(* Logix 5000 project; controller NSH_PLC2 vendor 1 type 14 code 167 rev 32.14; software revision 32.03; part 5 of 6 *)
(* tags used below, declared in another part *)
   AFI : BOOL;   // Always False
   AOI_MCC4_3E_ToPLC1 : E300ToMotor;
   AOI_MCC4_3G_ToPLC1 : E300ToMotor;
   AOI_MCC4_3J_ToPLC1 : E300ToMotor;
   AOI_MCC4_3L_ToPLC1 : E300ToMotor;
   AOI_MCC4_4A_ToPLC1 : E300ToMotor;
   AOI_MCC4_4C_ToPLC1 : E300ToMotor;
   AOI_MCC4_4E_ToPLC1 : E300ToMotor;
   AOI_MCC4_4G_ToPLC1 : E300ToMotor;
   AOI_MCC4_4J_ToPLC1 : E300ToMotor;
   AOI_MCC4_4L_ToPLC1 : E300ToMotor;
   AOI_MCC4_5A_ToPLC1 : E300ToMotor;
   AOI_MCC4_5C_ToPLC1 : E300ToMotor;
   AOI_PLC1_To_MCC2_10A : MotorToE300;
   AOI_PLC1_To_MCC2_10C : MotorToE300;
   AOI_PLC1_To_MCC2_10E : MotorToE300;
   AOI_PLC1_To_MCC2_10G : MotorToE300;
   AOI_PLC1_To_MCC2_10J : MotorToE300;
   AOI_PLC1_To_MCC2_10L : MotorToE300;
   AOI_PLC1_To_MCC2_11A : MotorToE300;
   AOI_PLC1_To_MCC2_11C : MotorToE300;
   AOI_PLC1_To_MCC2_11E : MotorToE300;
   AOI_PLC1_To_MCC2_11G : MotorToE300;
   AOI_PLC1_To_MCC2_11J : MotorToE300;
   AOI_PLC1_To_MCC2_11L : MotorToE300;
   AOI_PLC1_To_MCC2_12A : MotorToE300;
   AOI_PLC1_To_MCC2_12C : MotorToE300;
   AOI_PLC1_To_MCC2_12E : MotorToE300;
   AOI_PLC1_To_MCC2_12G : MotorToE300;
   AOI_PLC1_To_MCC2_12J : MotorToE300;
   AOI_PLC1_To_MCC2_12L : MotorToE300;
   AOI_PLC1_To_MCC2_13A : MotorToE300;
   AOI_PLC1_To_MCC2_13C : MotorToE300;
   AOI_PLC1_To_MCC2_13E : MotorToE300;
   AOI_PLC1_To_MCC2_13G : MotorToE300;
   AOI_PLC1_To_MCC2_13J : MotorToE300;
   AOI_PLC1_To_MCC2_14A : MotorToE300;
   AOI_PLC1_To_MCC2_14C : MotorToE300;
   AOI_PLC1_To_MCC2_14E : MotorToE300;
   AOI_PLC1_To_MCC2_14G : MotorToE300;
   AOI_PLC1_To_MCC2_14J : MotorToE300;
   AOI_PLC1_To_MCC2_14L : MotorToE300;
   AOI_PLC1_To_MCC2_15A : MotorToE300;
   AOI_PLC1_To_MCC2_15C : MotorToE300;
   AOI_PLC1_To_MCC2_15E : MotorToE300;
   AOI_PLC1_To_MCC2_15G : MotorToE300;
   AOI_PLC1_To_MCC2_15J : MotorToE300;
   AOI_PLC1_To_MCC2_15L : MotorToE300;
   AOI_PLC1_To_MCC2_16A : MotorToE300;
   AOI_PLC1_To_MCC2_16C : MotorToE300;
   AOI_PLC1_To_MCC2_16E : MotorToE300;
   AOI_PLC1_To_MCC2_16G : MotorToE300;
   AOI_PLC1_To_MCC2_16J : MotorToE300;
   AOI_PLC1_To_MCC2_16L : MotorToE300;
   AOI_PLC1_To_MCC2_17A : MotorToE300;
   AOI_PLC1_To_MCC2_17C : MotorToE300;
   AOI_PLC1_To_MCC2_17E : MotorToE300;
   AOI_PLC1_To_MCC2_17G : MotorToE300;
   AOI_PLC1_To_MCC2_17J : MotorToE300;
   AOI_PLC1_To_MCC2_18A : MotorToE300;
   AOI_PLC1_To_MCC2_18C : MotorToE300;
   AOI_PLC1_To_MCC2_18E : MotorToE300;
   AOI_PLC1_To_MCC2_18G : MotorToE300;
   AOI_PLC1_To_MCC2_18J : MotorToE300;
   AOI_PLC1_To_MCC2_18L : MotorToE300;
   AOI_PLC1_To_MCC2_19A : MotorToE300;
   AOI_PLC1_To_MCC2_19C : MotorToE300;
   AOI_PLC1_To_MCC2_19E : MotorToE300;
   AOI_PLC1_To_MCC2_19G : MotorToE300;
   AOI_PLC1_To_MCC2_19J : MotorToE300;
   AOI_PLC1_To_MCC2_19L : MotorToE300;
   AOI_PLC1_To_MCC2_20C : MotorToE300;
   AOI_PLC1_To_MCC2_20E : MotorToE300;
   AOI_PLC1_To_MCC2_20G : MotorToE300;
   AOI_PLC1_To_MCC2_20J : MotorToE300;
   AOI_PLC1_To_MCC2_21A : MotorToE300;
   AOI_PLC1_To_MCC2_21C : MotorToE300;
   AOI_PLC1_To_MCC2_21E : MotorToE300;
   AOI_PLC1_To_MCC2_21G : MotorToPF525;
   AOI_PLC1_To_MCC2_21K : MotorToPF525;
   AOI_PLC1_To_MCC2_2A : MotorToPF525;   // Motor From PLC1 to PF525 AOI
   AOI_PLC1_To_MCC2_2D : MotorToPF525;
   AOI_PLC1_To_MCC2_2G : MotorToPF525;
   AOI_PLC1_To_MCC2_2K : MotorToPF525;
   AOI_PLC1_To_MCC2_3A : MotorToE300;
   AOI_PLC1_To_MCC2_3C : MotorToE300;
   AOI_PLC1_To_MCC2_3E : MotorToE300;
   AOI_PLC1_To_MCC2_3G : MotorToE300;
   AOI_PLC1_To_MCC2_3J : MotorToE300;
   AOI_PLC1_To_MCC2_3L : MotorToE300;
   AOI_PLC1_To_MCC2_4A : MotorToE300;
   AOI_PLC1_To_MCC2_4C : MotorToE300;
   AOI_PLC1_To_MCC2_4E : MotorToE300;
   AOI_PLC1_To_MCC2_4G : MotorToE300;
   AOI_PLC1_To_MCC2_4J : MotorToE300;
   AOI_PLC1_To_MCC2_4L : MotorToE300;
   AOI_PLC1_To_MCC2_5A : MotorToE300;
   AOI_PLC1_To_MCC2_5C : MotorToE300;
   AOI_PLC1_To_MCC2_5E : MotorToE300;
   AOI_PLC1_To_MCC2_5G : MotorToE300;
   AOI_PLC1_To_MCC2_5J : MotorToE300;
   AOI_PLC1_To_MCC2_6A : MotorToE300;
   AOI_PLC1_To_MCC2_6C : MotorToE300;
   AOI_PLC1_To_MCC2_6E : MotorToE300;
   AOI_PLC1_To_MCC2_6G : MotorToE300;
   AOI_PLC1_To_MCC2_6J : MotorToE300;
   AOI_PLC1_To_MCC2_6L : MotorToE300;
   AOI_PLC1_To_MCC2_7A : MotorToE300;
   AOI_PLC1_To_MCC2_7D : MotorToE300;
   AOI_PLC1_To_MCC2_7G : MotorToE300;
   AOI_PLC1_To_MCC2_7K : MotorToE300;
   AOI_PLC1_To_MCC2_8B : MotorToE300;
   AOI_PLC1_To_MCC2_8D : MotorToE300;
   AOI_PLC1_To_MCC2_8F : MotorToE300;
   AOI_PLC1_To_MCC2_8H : MotorToE300;
   AOI_PLC1_To_MCC2_8K : MotorToE300;
   AOI_PLC1_To_MCC2_9D : MotorToE300;
   AOI_PLC1_To_MCC2_9F : MotorToE300;
   AOI_PLC1_To_MCC2_9H : MotorToPF525;
   AOI_PLC1_To_MCC3_2A : MotorToPF525;
   AOI_PLC1_To_MCC3_2D : MotorToPF525;
   AOI_PLC1_To_MCC3_2G : MotorToPF525;
   AOI_PLC1_To_MCC3_2K : MotorToPF525;
   AOI_PLC1_To_MCC3_3A : MotorToPF525;
   AOI_PLC1_To_MCC3_3D : MotorToPF525;
   AOI_PLC1_To_MCC3_3G : MotorToPF525;
   AOI_PLC1_To_MCC3_3K : MotorToPF525;
   AOI_PLC1_To_MCC3_4A : MotorToPF525;
   AOI_PLC1_To_MCC3_4D : MotorToPF525;
   AOI_PLC1_To_MCC3_4G : MotorToPF525;
   AOI_PLC1_To_MCC3_4K : MotorToPF525;
   AOI_PLC1_To_MCC3_5A : MotorToPF525;
   AOI_PLC1_To_MCC3_5D : MotorToPF525;
   AOI_PLC1_To_MCC3_5G : MotorToPF525;
   AOI_PLC1_To_MCC3_5K : MotorToPF525;
   AOI_PLC1_To_MCC3_6A : MotorToPF525;
   AOI_PLC1_To_MCC3_6D : MotorToPF525;
   AOI_PLC1_To_MCC3_6G : MotorToE300;
   AOI_PLC1_To_MCC3_6J : MotorToE300;
   Const_4000_Hex : INT;   // Constant #16:4000, Entry Status Communicating
   GSV_EntryStatus : INT;   // GSV Entry Status, shold be #16:4000
   MCC4_3E_CommsOK : BOOL;   // Communications with AOP OK
   MCC4_3G_CommsOK : BOOL;   // Communications with AOP OK
   MCC4_3J_CommsOK : BOOL;   // Communications with AOP OK
   MCC4_3L_CommsOK : BOOL;   // Communications with AOP OK
   MCC4_4A_CommsOK : BOOL;   // Communications with AOP OK
   MCC4_4C_CommsOK : BOOL;   // Communications with AOP OK
   MCC4_4E_CommsOK : BOOL;   // Communications with AOP OK
   MCC4_4G_CommsOK : BOOL;   // Communications with AOP OK
   MCC4_4J_CommsOK : BOOL;   // Communications with AOP OK
   MCC4_4L_CommsOK : BOOL;   // Communications with AOP OK
   MCC4_5A_CommsOK : BOOL;   // Communications with AOP OK
   MCC4_5C_CommsOK : BOOL;   // Communications with AOP OK
   MotorsControlTag : MotorsControlUDT;   // Only Instance of UDT
   MotorsStatusTag : MotorsStatusUDT;   // Only Instance of UDT
   MSG_ReadSpacing_T : TIMER;   // Read MCC2 & MCC3 Motor Commands From PLC1 Spacing Timer
   OKToRunMotors : BOOL;   // Messages from PLC1 Ok, OK to run
   ReadMotorError_CTR : COUNTER;   // Read Message form PLC1 Error Counter
   ReadMotorsFromPLC1 : MESSAGE;   // Read from PLC1, MotorsToPLC2
   ReadMotorsFromPLC1_DOS : BOOL;   // Read Motors from PLC1 Done One Shot
(* MainProgram, continued *)

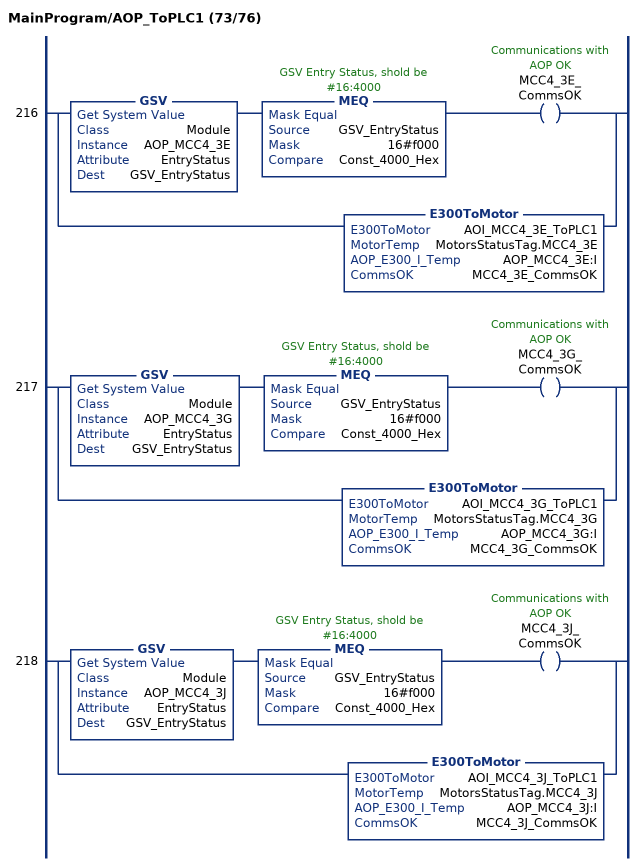
   216: [GSV(Module,AOP_MCC4_3E,EntryStatus,GSV_EntryStatus) MEQ(GSV_EntryStatus,16#f000,Const_4000_Hex) OTE(MCC4_3E_CommsOK) ,E300ToMotor(AOI_MCC4_3E_ToPLC1,MotorsStatusTag.MCC4_3E,AOP_MCC4_3E:I,MCC4_3E_CommsOK) ];
   217: [GSV(Module,AOP_MCC4_3G,EntryStatus,GSV_EntryStatus) MEQ(GSV_EntryStatus,16#f000,Const_4000_Hex) OTE(MCC4_3G_CommsOK) ,E300ToMotor(AOI_MCC4_3G_ToPLC1,MotorsStatusTag.MCC4_3G,AOP_MCC4_3G:I,MCC4_3G_CommsOK) ];
   218: [GSV(Module,AOP_MCC4_3J,EntryStatus,GSV_EntryStatus) MEQ(GSV_EntryStatus,16#f000,Const_4000_Hex) OTE(MCC4_3J_CommsOK) ,E300ToMotor(AOI_MCC4_3J_ToPLC1,MotorsStatusTag.MCC4_3J,AOP_MCC4_3J:I,MCC4_3J_CommsOK) ];
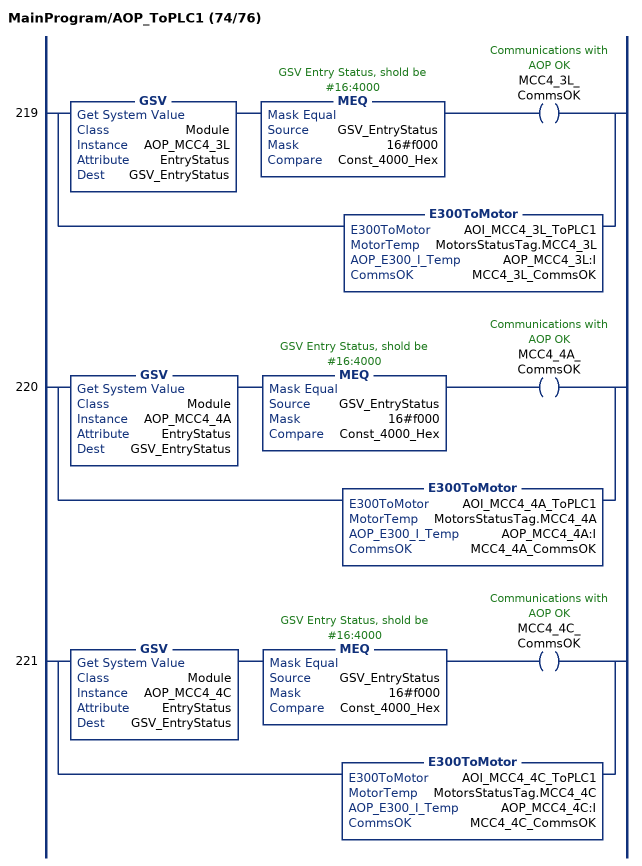
   219: [GSV(Module,AOP_MCC4_3L,EntryStatus,GSV_EntryStatus) MEQ(GSV_EntryStatus,16#f000,Const_4000_Hex) OTE(MCC4_3L_CommsOK) ,E300ToMotor(AOI_MCC4_3L_ToPLC1,MotorsStatusTag.MCC4_3L,AOP_MCC4_3L:I,MCC4_3L_CommsOK) ];
   220: [GSV(Module,AOP_MCC4_4A,EntryStatus,GSV_EntryStatus) MEQ(GSV_EntryStatus,16#f000,Const_4000_Hex) OTE(MCC4_4A_CommsOK) ,E300ToMotor(AOI_MCC4_4A_ToPLC1,MotorsStatusTag.MCC4_4A,AOP_MCC4_4A:I,MCC4_4A_CommsOK) ];
   221: [GSV(Module,AOP_MCC4_4C,EntryStatus,GSV_EntryStatus) MEQ(GSV_EntryStatus,16#f000,Const_4000_Hex) OTE(MCC4_4C_CommsOK) ,E300ToMotor(AOI_MCC4_4C_ToPLC1,MotorsStatusTag.MCC4_4C,AOP_MCC4_4C:I,MCC4_4C_CommsOK) ];
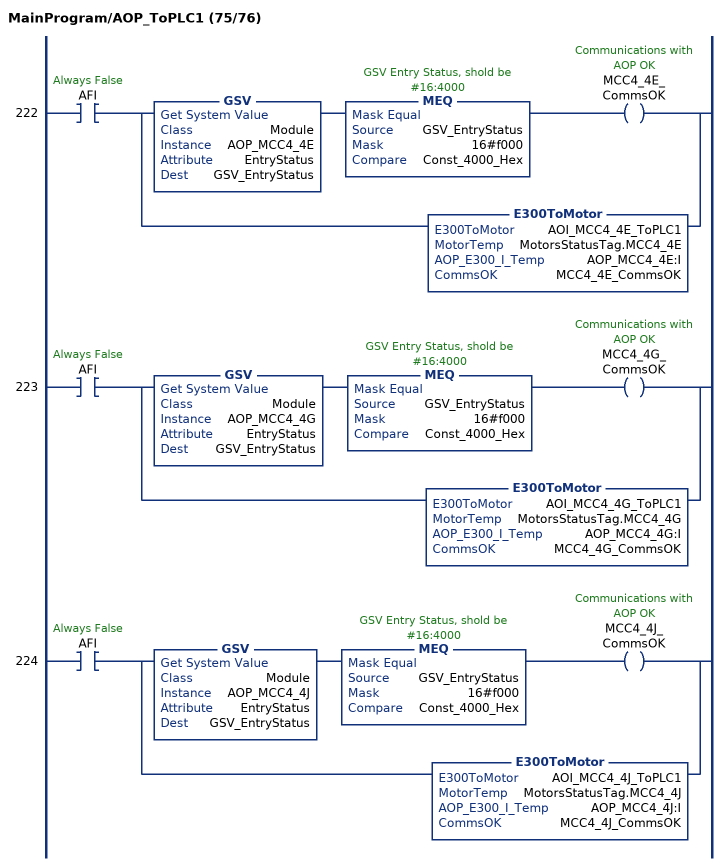
   222: XIC(AFI)[GSV(Module,AOP_MCC4_4E,EntryStatus,GSV_EntryStatus) MEQ(GSV_EntryStatus,16#f000,Const_4000_Hex) OTE(MCC4_4E_CommsOK) ,E300ToMotor(AOI_MCC4_4E_ToPLC1,MotorsStatusTag.MCC4_4E,AOP_MCC4_4E:I,MCC4_4E_CommsOK) ];
   223: XIC(AFI)[GSV(Module,AOP_MCC4_4G,EntryStatus,GSV_EntryStatus) MEQ(GSV_EntryStatus,16#f000,Const_4000_Hex) OTE(MCC4_4G_CommsOK) ,E300ToMotor(AOI_MCC4_4G_ToPLC1,MotorsStatusTag.MCC4_4G,AOP_MCC4_4G:I,MCC4_4G_CommsOK) ];
   224: XIC(AFI)[GSV(Module,AOP_MCC4_4J,EntryStatus,GSV_EntryStatus) MEQ(GSV_EntryStatus,16#f000,Const_4000_Hex) OTE(MCC4_4J_CommsOK) ,E300ToMotor(AOI_MCC4_4J_ToPLC1,MotorsStatusTag.MCC4_4J,AOP_MCC4_4J:I,MCC4_4J_CommsOK) ];
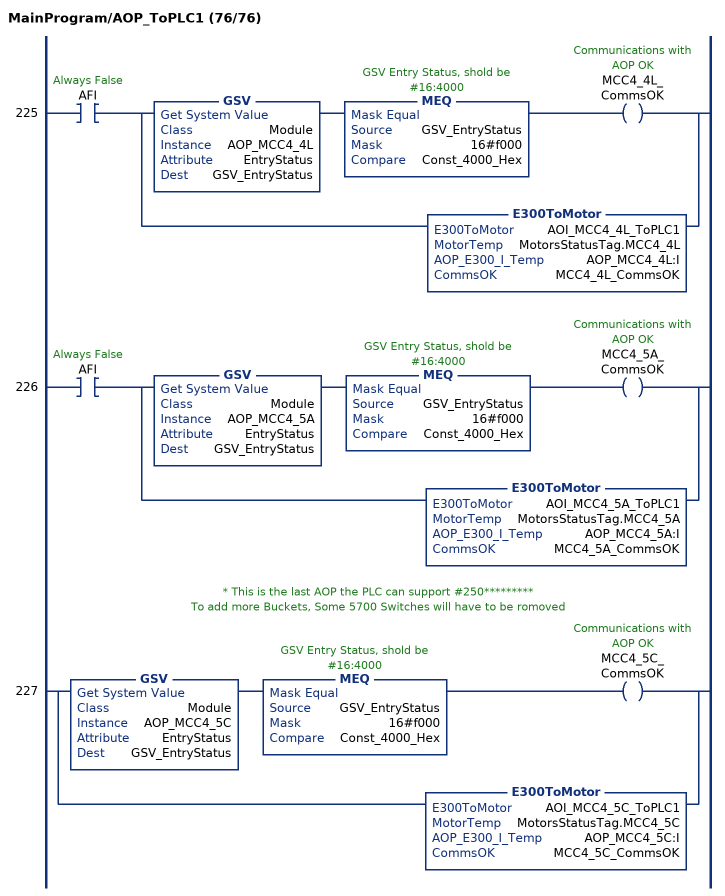
   225: XIC(AFI)[GSV(Module,AOP_MCC4_4L,EntryStatus,GSV_EntryStatus) MEQ(GSV_EntryStatus,16#f000,Const_4000_Hex) OTE(MCC4_4L_CommsOK) ,E300ToMotor(AOI_MCC4_4L_ToPLC1,MotorsStatusTag.MCC4_4L,AOP_MCC4_4L:I,MCC4_4L_CommsOK) ];
   226: XIC(AFI)[GSV(Module,AOP_MCC4_5A,EntryStatus,GSV_EntryStatus) MEQ(GSV_EntryStatus,16#f000,Const_4000_Hex) OTE(MCC4_5A_CommsOK) ,E300ToMotor(AOI_MCC4_5A_ToPLC1,MotorsStatusTag.MCC4_5A,AOP_MCC4_5A:I,MCC4_5A_CommsOK) ];
   // * This is the last AOP the PLC can support #250*********
   // To add more Buckets, Some 5700 Switches will have to be romoved
   227: [GSV(Module,AOP_MCC4_5C,EntryStatus,GSV_EntryStatus) MEQ(GSV_EntryStatus,16#f000,Const_4000_Hex) OTE(MCC4_5C_CommsOK) ,E300ToMotor(AOI_MCC4_5C_ToPLC1,MotorsStatusTag.MCC4_5C,AOP_MCC4_5C:I,MCC4_5C_CommsOK) ];
END_ROUTINE

ROUTINE MainRoutine   (* ladder *)
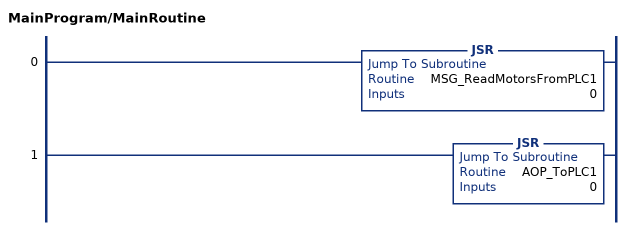
   0: JSR(MSG_ReadMotorsFromPLC1,0);
   1: JSR(AOP_ToPLC1,0);
END_ROUTINE

ROUTINE MSG_ReadMotorsFromPLC1   (* ladder *)
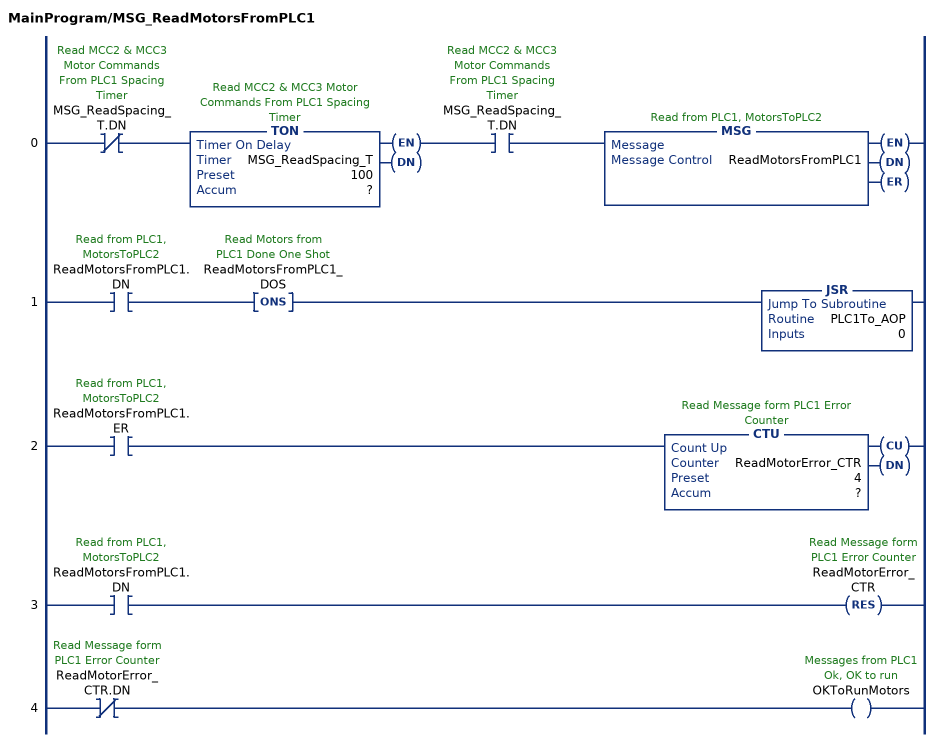
   0: XIO(MSG_ReadSpacing_T.DN)TON(MSG_ReadSpacing_T,?,?)XIC(MSG_ReadSpacing_T.DN)MSG(ReadMotorsFromPLC1);
   1: XIC(ReadMotorsFromPLC1.DN)ONS(ReadMotorsFromPLC1_DOS)JSR(PLC1To_AOP,0);
   2: XIC(ReadMotorsFromPLC1.ER)CTU(ReadMotorError_CTR,?,?);
   3: XIC(ReadMotorsFromPLC1.DN)RES(ReadMotorError_CTR);
   4: XIO(ReadMotorError_CTR.DN)OTE(OKToRunMotors);
END_ROUTINE

ROUTINE PLC1To_AOP   (* ladder *)
// Send Command Data from PLC#1 to AOPs
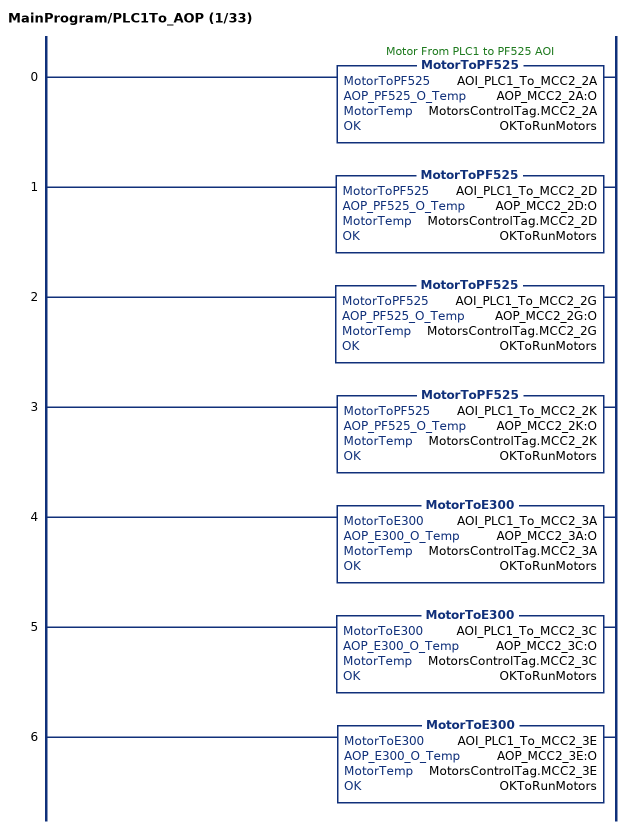
   0: MotorToPF525(AOI_PLC1_To_MCC2_2A,AOP_MCC2_2A:O,MotorsControlTag.MCC2_2A,OKToRunMotors);
   1: MotorToPF525(AOI_PLC1_To_MCC2_2D,AOP_MCC2_2D:O,MotorsControlTag.MCC2_2D,OKToRunMotors);
   2: MotorToPF525(AOI_PLC1_To_MCC2_2G,AOP_MCC2_2G:O,MotorsControlTag.MCC2_2G,OKToRunMotors);
   3: MotorToPF525(AOI_PLC1_To_MCC2_2K,AOP_MCC2_2K:O,MotorsControlTag.MCC2_2K,OKToRunMotors);
   4: MotorToE300(AOI_PLC1_To_MCC2_3A,AOP_MCC2_3A:O,MotorsControlTag.MCC2_3A,OKToRunMotors);
   5: MotorToE300(AOI_PLC1_To_MCC2_3C,AOP_MCC2_3C:O,MotorsControlTag.MCC2_3C,OKToRunMotors);
   6: MotorToE300(AOI_PLC1_To_MCC2_3E,AOP_MCC2_3E:O,MotorsControlTag.MCC2_3E,OKToRunMotors);
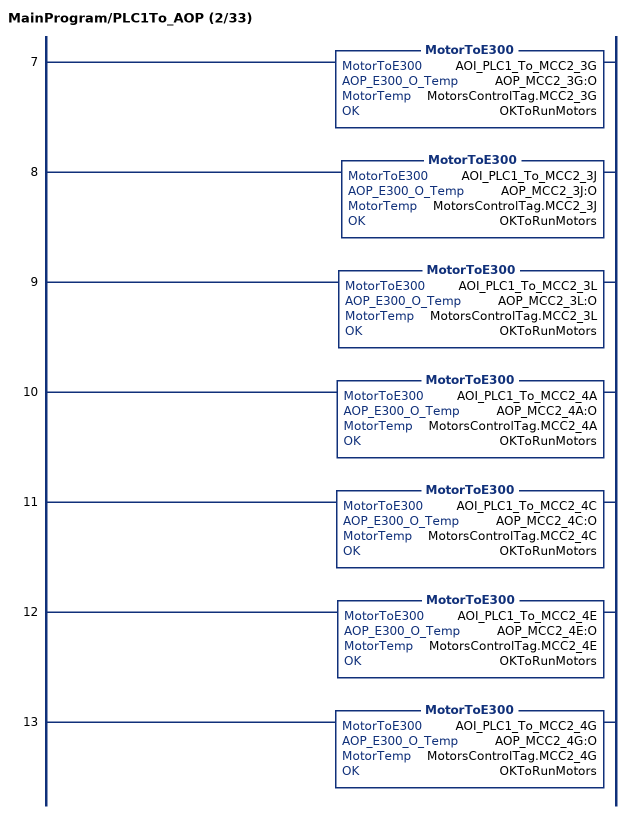
   7: MotorToE300(AOI_PLC1_To_MCC2_3G,AOP_MCC2_3G:O,MotorsControlTag.MCC2_3G,OKToRunMotors);
   8: MotorToE300(AOI_PLC1_To_MCC2_3J,AOP_MCC2_3J:O,MotorsControlTag.MCC2_3J,OKToRunMotors);
   9: MotorToE300(AOI_PLC1_To_MCC2_3L,AOP_MCC2_3L:O,MotorsControlTag.MCC2_3L,OKToRunMotors);
   10: MotorToE300(AOI_PLC1_To_MCC2_4A,AOP_MCC2_4A:O,MotorsControlTag.MCC2_4A,OKToRunMotors);
   11: MotorToE300(AOI_PLC1_To_MCC2_4C,AOP_MCC2_4C:O,MotorsControlTag.MCC2_4C,OKToRunMotors);
   12: MotorToE300(AOI_PLC1_To_MCC2_4E,AOP_MCC2_4E:O,MotorsControlTag.MCC2_4E,OKToRunMotors);
   13: MotorToE300(AOI_PLC1_To_MCC2_4G,AOP_MCC2_4G:O,MotorsControlTag.MCC2_4G,OKToRunMotors);
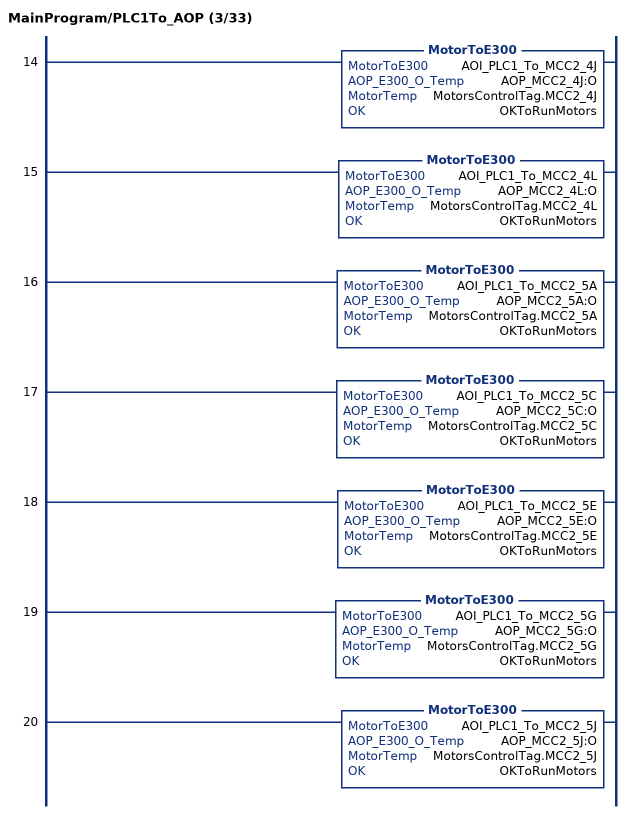
   14: MotorToE300(AOI_PLC1_To_MCC2_4J,AOP_MCC2_4J:O,MotorsControlTag.MCC2_4J,OKToRunMotors);
   15: MotorToE300(AOI_PLC1_To_MCC2_4L,AOP_MCC2_4L:O,MotorsControlTag.MCC2_4L,OKToRunMotors);
   16: MotorToE300(AOI_PLC1_To_MCC2_5A,AOP_MCC2_5A:O,MotorsControlTag.MCC2_5A,OKToRunMotors);
   17: MotorToE300(AOI_PLC1_To_MCC2_5C,AOP_MCC2_5C:O,MotorsControlTag.MCC2_5C,OKToRunMotors);
   18: MotorToE300(AOI_PLC1_To_MCC2_5E,AOP_MCC2_5E:O,MotorsControlTag.MCC2_5E,OKToRunMotors);
   19: MotorToE300(AOI_PLC1_To_MCC2_5G,AOP_MCC2_5G:O,MotorsControlTag.MCC2_5G,OKToRunMotors);
   20: MotorToE300(AOI_PLC1_To_MCC2_5J,AOP_MCC2_5J:O,MotorsControlTag.MCC2_5J,OKToRunMotors);
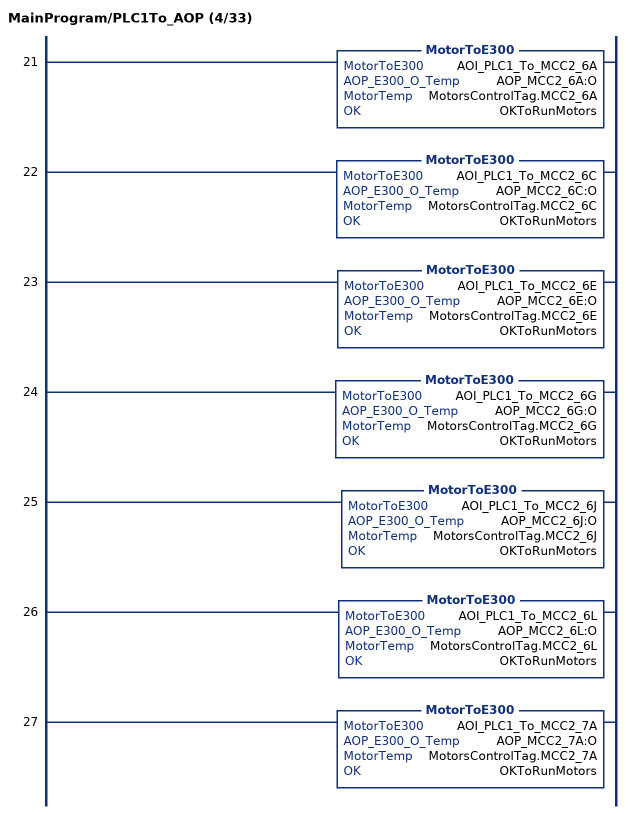
   21: MotorToE300(AOI_PLC1_To_MCC2_6A,AOP_MCC2_6A:O,MotorsControlTag.MCC2_6A,OKToRunMotors);
   22: MotorToE300(AOI_PLC1_To_MCC2_6C,AOP_MCC2_6C:O,MotorsControlTag.MCC2_6C,OKToRunMotors);
   23: MotorToE300(AOI_PLC1_To_MCC2_6E,AOP_MCC2_6E:O,MotorsControlTag.MCC2_6E,OKToRunMotors);
   24: MotorToE300(AOI_PLC1_To_MCC2_6G,AOP_MCC2_6G:O,MotorsControlTag.MCC2_6G,OKToRunMotors);
   25: MotorToE300(AOI_PLC1_To_MCC2_6J,AOP_MCC2_6J:O,MotorsControlTag.MCC2_6J,OKToRunMotors);
   26: MotorToE300(AOI_PLC1_To_MCC2_6L,AOP_MCC2_6L:O,MotorsControlTag.MCC2_6L,OKToRunMotors);
   27: MotorToE300(AOI_PLC1_To_MCC2_7A,AOP_MCC2_7A:O,MotorsControlTag.MCC2_7A,OKToRunMotors);
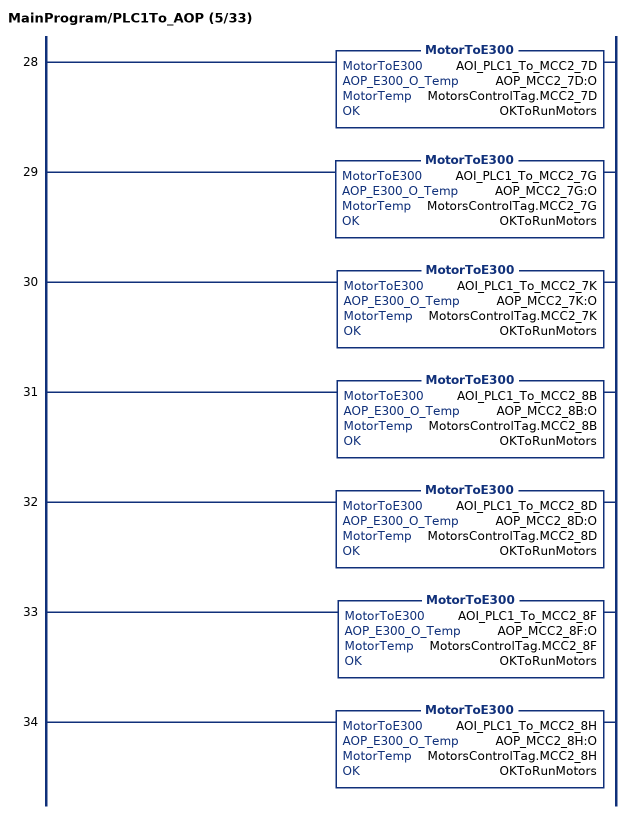
   28: MotorToE300(AOI_PLC1_To_MCC2_7D,AOP_MCC2_7D:O,MotorsControlTag.MCC2_7D,OKToRunMotors);
   29: MotorToE300(AOI_PLC1_To_MCC2_7G,AOP_MCC2_7G:O,MotorsControlTag.MCC2_7G,OKToRunMotors);
   30: MotorToE300(AOI_PLC1_To_MCC2_7K,AOP_MCC2_7K:O,MotorsControlTag.MCC2_7K,OKToRunMotors);
   31: MotorToE300(AOI_PLC1_To_MCC2_8B,AOP_MCC2_8B:O,MotorsControlTag.MCC2_8B,OKToRunMotors);
   32: MotorToE300(AOI_PLC1_To_MCC2_8D,AOP_MCC2_8D:O,MotorsControlTag.MCC2_8D,OKToRunMotors);
   33: MotorToE300(AOI_PLC1_To_MCC2_8F,AOP_MCC2_8F:O,MotorsControlTag.MCC2_8F,OKToRunMotors);
   34: MotorToE300(AOI_PLC1_To_MCC2_8H,AOP_MCC2_8H:O,MotorsControlTag.MCC2_8H,OKToRunMotors);
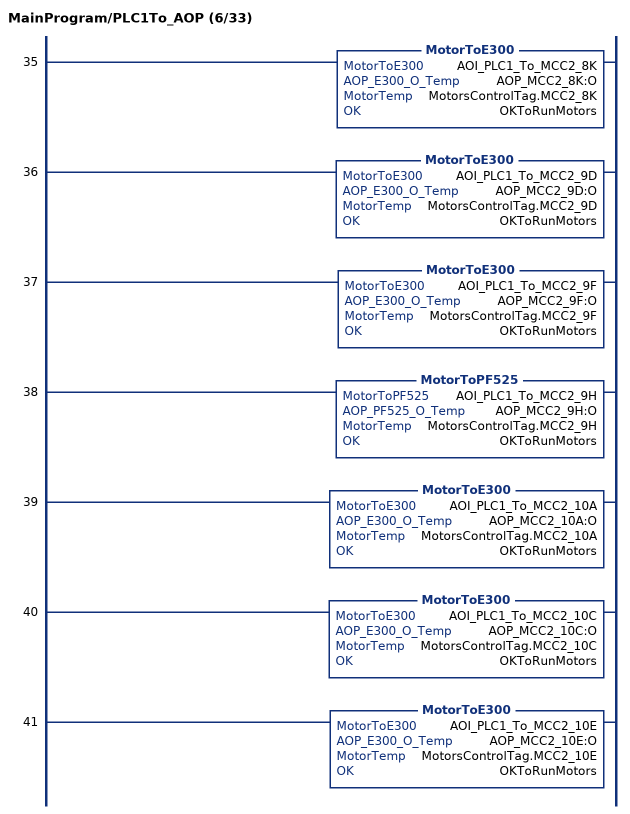
   35: MotorToE300(AOI_PLC1_To_MCC2_8K,AOP_MCC2_8K:O,MotorsControlTag.MCC2_8K,OKToRunMotors);
   36: MotorToE300(AOI_PLC1_To_MCC2_9D,AOP_MCC2_9D:O,MotorsControlTag.MCC2_9D,OKToRunMotors);
   37: MotorToE300(AOI_PLC1_To_MCC2_9F,AOP_MCC2_9F:O,MotorsControlTag.MCC2_9F,OKToRunMotors);
   38: MotorToPF525(AOI_PLC1_To_MCC2_9H,AOP_MCC2_9H:O,MotorsControlTag.MCC2_9H,OKToRunMotors);
   39: MotorToE300(AOI_PLC1_To_MCC2_10A,AOP_MCC2_10A:O,MotorsControlTag.MCC2_10A,OKToRunMotors);
   40: MotorToE300(AOI_PLC1_To_MCC2_10C,AOP_MCC2_10C:O,MotorsControlTag.MCC2_10C,OKToRunMotors);
   41: MotorToE300(AOI_PLC1_To_MCC2_10E,AOP_MCC2_10E:O,MotorsControlTag.MCC2_10E,OKToRunMotors);
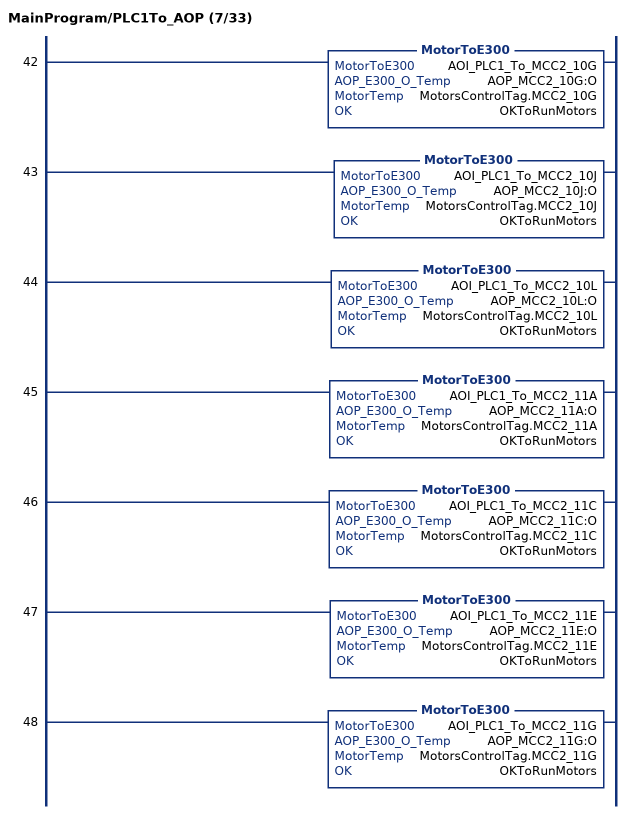
   42: MotorToE300(AOI_PLC1_To_MCC2_10G,AOP_MCC2_10G:O,MotorsControlTag.MCC2_10G,OKToRunMotors);
   43: MotorToE300(AOI_PLC1_To_MCC2_10J,AOP_MCC2_10J:O,MotorsControlTag.MCC2_10J,OKToRunMotors);
   44: MotorToE300(AOI_PLC1_To_MCC2_10L,AOP_MCC2_10L:O,MotorsControlTag.MCC2_10L,OKToRunMotors);
   45: MotorToE300(AOI_PLC1_To_MCC2_11A,AOP_MCC2_11A:O,MotorsControlTag.MCC2_11A,OKToRunMotors);
   46: MotorToE300(AOI_PLC1_To_MCC2_11C,AOP_MCC2_11C:O,MotorsControlTag.MCC2_11C,OKToRunMotors);
   47: MotorToE300(AOI_PLC1_To_MCC2_11E,AOP_MCC2_11E:O,MotorsControlTag.MCC2_11E,OKToRunMotors);
   48: MotorToE300(AOI_PLC1_To_MCC2_11G,AOP_MCC2_11G:O,MotorsControlTag.MCC2_11G,OKToRunMotors);
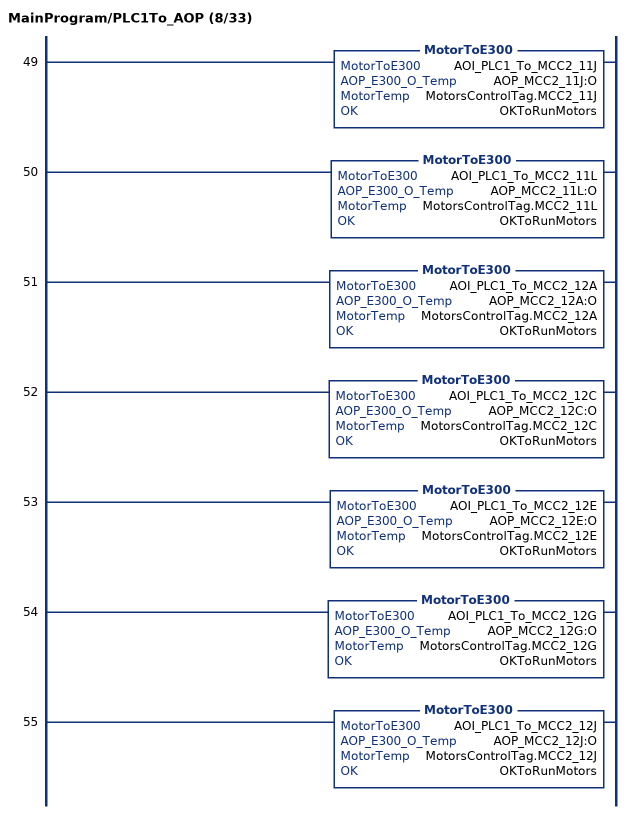
   49: MotorToE300(AOI_PLC1_To_MCC2_11J,AOP_MCC2_11J:O,MotorsControlTag.MCC2_11J,OKToRunMotors);
   50: MotorToE300(AOI_PLC1_To_MCC2_11L,AOP_MCC2_11L:O,MotorsControlTag.MCC2_11L,OKToRunMotors);
   51: MotorToE300(AOI_PLC1_To_MCC2_12A,AOP_MCC2_12A:O,MotorsControlTag.MCC2_12A,OKToRunMotors);
   52: MotorToE300(AOI_PLC1_To_MCC2_12C,AOP_MCC2_12C:O,MotorsControlTag.MCC2_12C,OKToRunMotors);
   53: MotorToE300(AOI_PLC1_To_MCC2_12E,AOP_MCC2_12E:O,MotorsControlTag.MCC2_12E,OKToRunMotors);
   54: MotorToE300(AOI_PLC1_To_MCC2_12G,AOP_MCC2_12G:O,MotorsControlTag.MCC2_12G,OKToRunMotors);
   55: MotorToE300(AOI_PLC1_To_MCC2_12J,AOP_MCC2_12J:O,MotorsControlTag.MCC2_12J,OKToRunMotors);
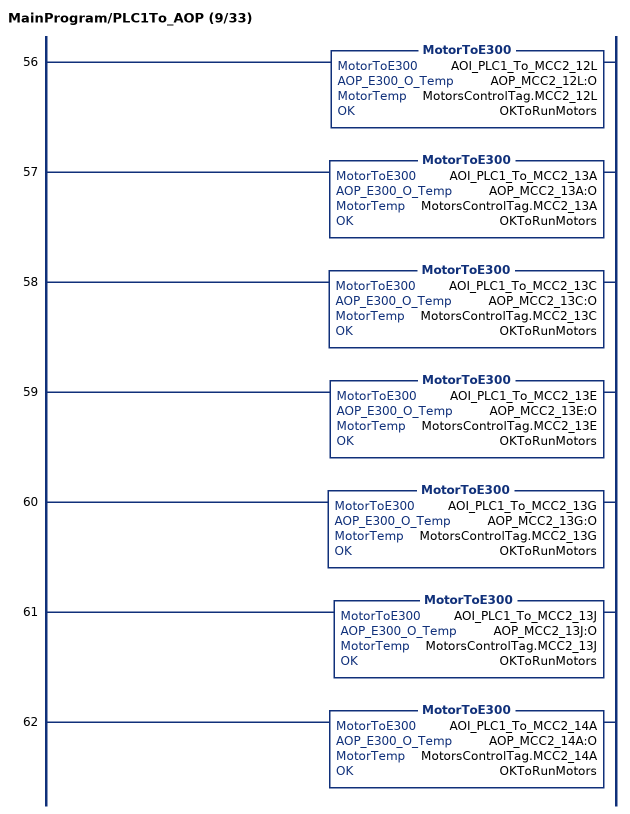
   56: MotorToE300(AOI_PLC1_To_MCC2_12L,AOP_MCC2_12L:O,MotorsControlTag.MCC2_12L,OKToRunMotors);
   57: MotorToE300(AOI_PLC1_To_MCC2_13A,AOP_MCC2_13A:O,MotorsControlTag.MCC2_13A,OKToRunMotors);
   58: MotorToE300(AOI_PLC1_To_MCC2_13C,AOP_MCC2_13C:O,MotorsControlTag.MCC2_13C,OKToRunMotors);
   59: MotorToE300(AOI_PLC1_To_MCC2_13E,AOP_MCC2_13E:O,MotorsControlTag.MCC2_13E,OKToRunMotors);
   60: MotorToE300(AOI_PLC1_To_MCC2_13G,AOP_MCC2_13G:O,MotorsControlTag.MCC2_13G,OKToRunMotors);
   61: MotorToE300(AOI_PLC1_To_MCC2_13J,AOP_MCC2_13J:O,MotorsControlTag.MCC2_13J,OKToRunMotors);
   62: MotorToE300(AOI_PLC1_To_MCC2_14A,AOP_MCC2_14A:O,MotorsControlTag.MCC2_14A,OKToRunMotors);
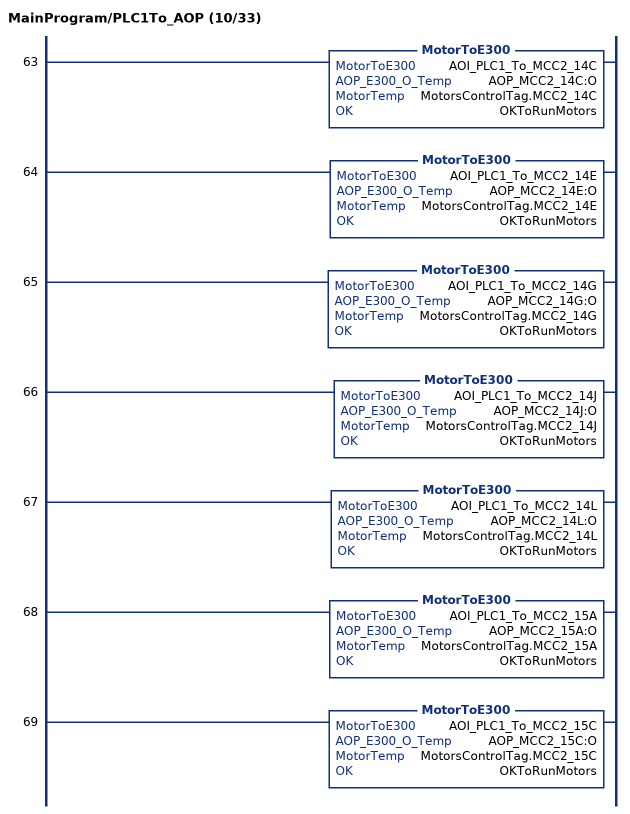
   63: MotorToE300(AOI_PLC1_To_MCC2_14C,AOP_MCC2_14C:O,MotorsControlTag.MCC2_14C,OKToRunMotors);
   64: MotorToE300(AOI_PLC1_To_MCC2_14E,AOP_MCC2_14E:O,MotorsControlTag.MCC2_14E,OKToRunMotors);
   65: MotorToE300(AOI_PLC1_To_MCC2_14G,AOP_MCC2_14G:O,MotorsControlTag.MCC2_14G,OKToRunMotors);
   66: MotorToE300(AOI_PLC1_To_MCC2_14J,AOP_MCC2_14J:O,MotorsControlTag.MCC2_14J,OKToRunMotors);
   67: MotorToE300(AOI_PLC1_To_MCC2_14L,AOP_MCC2_14L:O,MotorsControlTag.MCC2_14L,OKToRunMotors);
   68: MotorToE300(AOI_PLC1_To_MCC2_15A,AOP_MCC2_15A:O,MotorsControlTag.MCC2_15A,OKToRunMotors);
   69: MotorToE300(AOI_PLC1_To_MCC2_15C,AOP_MCC2_15C:O,MotorsControlTag.MCC2_15C,OKToRunMotors);
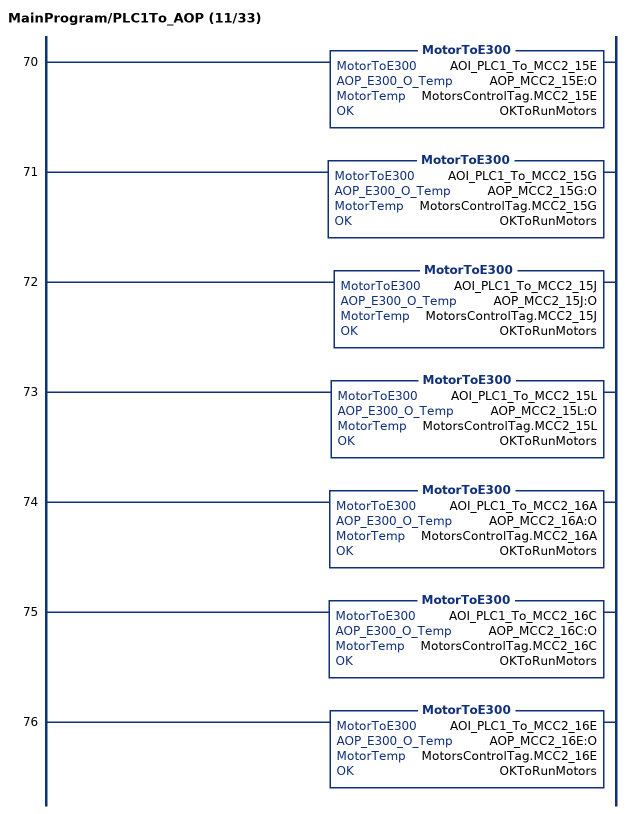
   70: MotorToE300(AOI_PLC1_To_MCC2_15E,AOP_MCC2_15E:O,MotorsControlTag.MCC2_15E,OKToRunMotors);
   71: MotorToE300(AOI_PLC1_To_MCC2_15G,AOP_MCC2_15G:O,MotorsControlTag.MCC2_15G,OKToRunMotors);
   72: MotorToE300(AOI_PLC1_To_MCC2_15J,AOP_MCC2_15J:O,MotorsControlTag.MCC2_15J,OKToRunMotors);
   73: MotorToE300(AOI_PLC1_To_MCC2_15L,AOP_MCC2_15L:O,MotorsControlTag.MCC2_15L,OKToRunMotors);
   74: MotorToE300(AOI_PLC1_To_MCC2_16A,AOP_MCC2_16A:O,MotorsControlTag.MCC2_16A,OKToRunMotors);
   75: MotorToE300(AOI_PLC1_To_MCC2_16C,AOP_MCC2_16C:O,MotorsControlTag.MCC2_16C,OKToRunMotors);
   76: MotorToE300(AOI_PLC1_To_MCC2_16E,AOP_MCC2_16E:O,MotorsControlTag.MCC2_16E,OKToRunMotors);
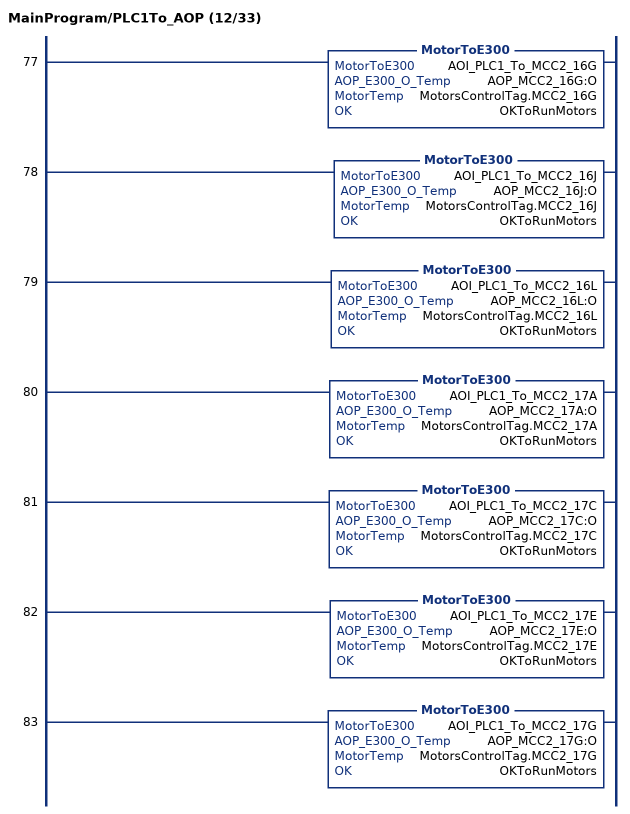
   77: MotorToE300(AOI_PLC1_To_MCC2_16G,AOP_MCC2_16G:O,MotorsControlTag.MCC2_16G,OKToRunMotors);
   78: MotorToE300(AOI_PLC1_To_MCC2_16J,AOP_MCC2_16J:O,MotorsControlTag.MCC2_16J,OKToRunMotors);
   79: MotorToE300(AOI_PLC1_To_MCC2_16L,AOP_MCC2_16L:O,MotorsControlTag.MCC2_16L,OKToRunMotors);
   80: MotorToE300(AOI_PLC1_To_MCC2_17A,AOP_MCC2_17A:O,MotorsControlTag.MCC2_17A,OKToRunMotors);
   81: MotorToE300(AOI_PLC1_To_MCC2_17C,AOP_MCC2_17C:O,MotorsControlTag.MCC2_17C,OKToRunMotors);
   82: MotorToE300(AOI_PLC1_To_MCC2_17E,AOP_MCC2_17E:O,MotorsControlTag.MCC2_17E,OKToRunMotors);
   83: MotorToE300(AOI_PLC1_To_MCC2_17G,AOP_MCC2_17G:O,MotorsControlTag.MCC2_17G,OKToRunMotors);
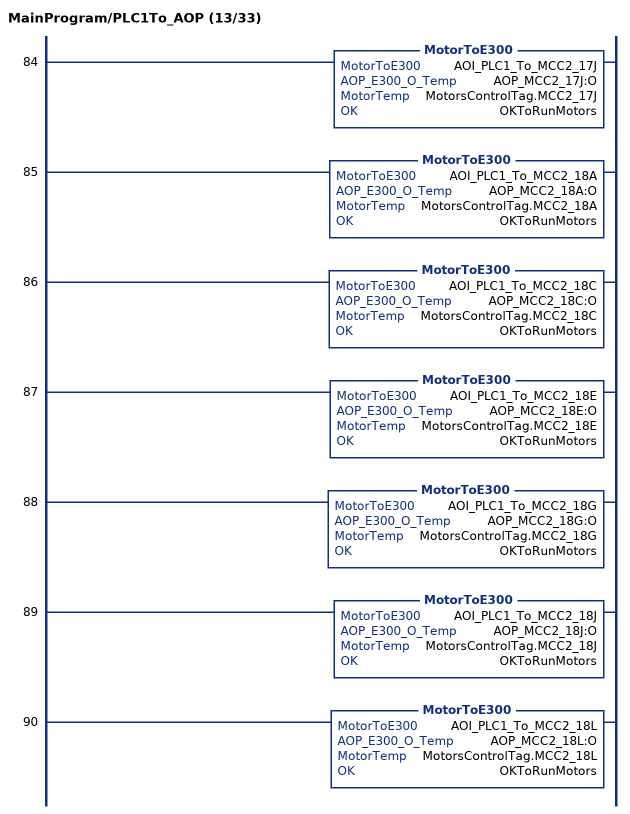
   84: MotorToE300(AOI_PLC1_To_MCC2_17J,AOP_MCC2_17J:O,MotorsControlTag.MCC2_17J,OKToRunMotors);
   85: MotorToE300(AOI_PLC1_To_MCC2_18A,AOP_MCC2_18A:O,MotorsControlTag.MCC2_18A,OKToRunMotors);
   86: MotorToE300(AOI_PLC1_To_MCC2_18C,AOP_MCC2_18C:O,MotorsControlTag.MCC2_18C,OKToRunMotors);
   87: MotorToE300(AOI_PLC1_To_MCC2_18E,AOP_MCC2_18E:O,MotorsControlTag.MCC2_18E,OKToRunMotors);
   88: MotorToE300(AOI_PLC1_To_MCC2_18G,AOP_MCC2_18G:O,MotorsControlTag.MCC2_18G,OKToRunMotors);
   89: MotorToE300(AOI_PLC1_To_MCC2_18J,AOP_MCC2_18J:O,MotorsControlTag.MCC2_18J,OKToRunMotors);
   90: MotorToE300(AOI_PLC1_To_MCC2_18L,AOP_MCC2_18L:O,MotorsControlTag.MCC2_18L,OKToRunMotors);
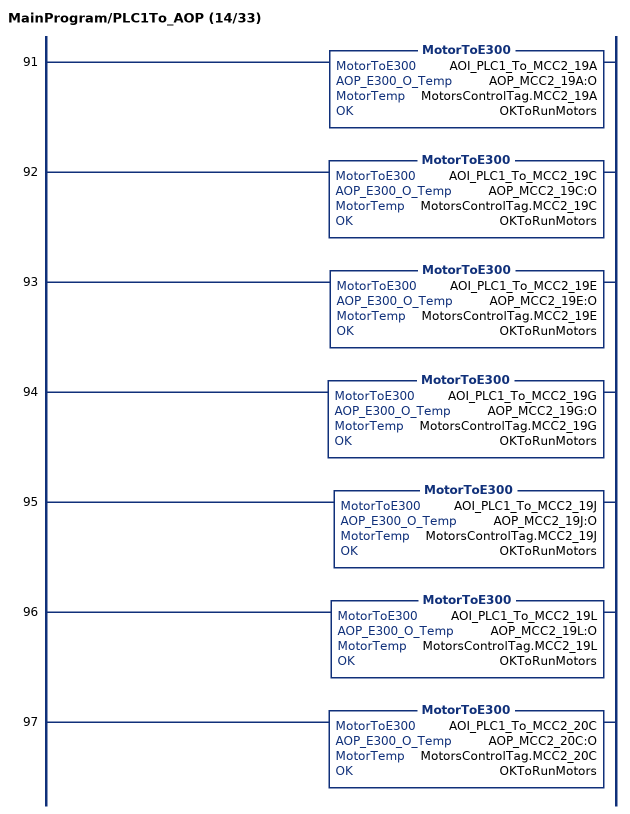
   91: MotorToE300(AOI_PLC1_To_MCC2_19A,AOP_MCC2_19A:O,MotorsControlTag.MCC2_19A,OKToRunMotors);
   92: MotorToE300(AOI_PLC1_To_MCC2_19C,AOP_MCC2_19C:O,MotorsControlTag.MCC2_19C,OKToRunMotors);
   93: MotorToE300(AOI_PLC1_To_MCC2_19E,AOP_MCC2_19E:O,MotorsControlTag.MCC2_19E,OKToRunMotors);
   94: MotorToE300(AOI_PLC1_To_MCC2_19G,AOP_MCC2_19G:O,MotorsControlTag.MCC2_19G,OKToRunMotors);
   95: MotorToE300(AOI_PLC1_To_MCC2_19J,AOP_MCC2_19J:O,MotorsControlTag.MCC2_19J,OKToRunMotors);
   96: MotorToE300(AOI_PLC1_To_MCC2_19L,AOP_MCC2_19L:O,MotorsControlTag.MCC2_19L,OKToRunMotors);
   97: MotorToE300(AOI_PLC1_To_MCC2_20C,AOP_MCC2_20C:O,MotorsControlTag.MCC2_20C,OKToRunMotors);
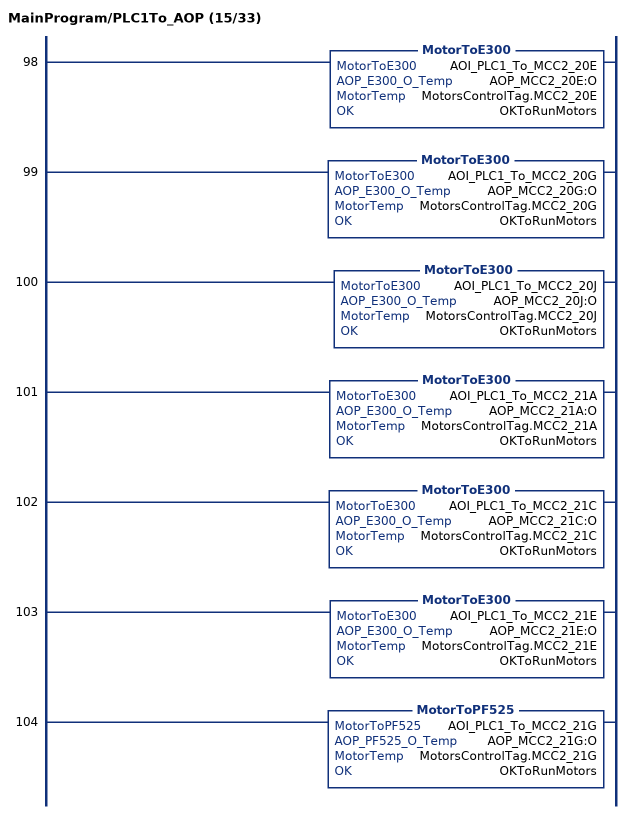
   98: MotorToE300(AOI_PLC1_To_MCC2_20E,AOP_MCC2_20E:O,MotorsControlTag.MCC2_20E,OKToRunMotors);
   99: MotorToE300(AOI_PLC1_To_MCC2_20G,AOP_MCC2_20G:O,MotorsControlTag.MCC2_20G,OKToRunMotors);
   100: MotorToE300(AOI_PLC1_To_MCC2_20J,AOP_MCC2_20J:O,MotorsControlTag.MCC2_20J,OKToRunMotors);
   101: MotorToE300(AOI_PLC1_To_MCC2_21A,AOP_MCC2_21A:O,MotorsControlTag.MCC2_21A,OKToRunMotors);
   102: MotorToE300(AOI_PLC1_To_MCC2_21C,AOP_MCC2_21C:O,MotorsControlTag.MCC2_21C,OKToRunMotors);
   103: MotorToE300(AOI_PLC1_To_MCC2_21E,AOP_MCC2_21E:O,MotorsControlTag.MCC2_21E,OKToRunMotors);
   104: MotorToPF525(AOI_PLC1_To_MCC2_21G,AOP_MCC2_21G:O,MotorsControlTag.MCC2_21G,OKToRunMotors);
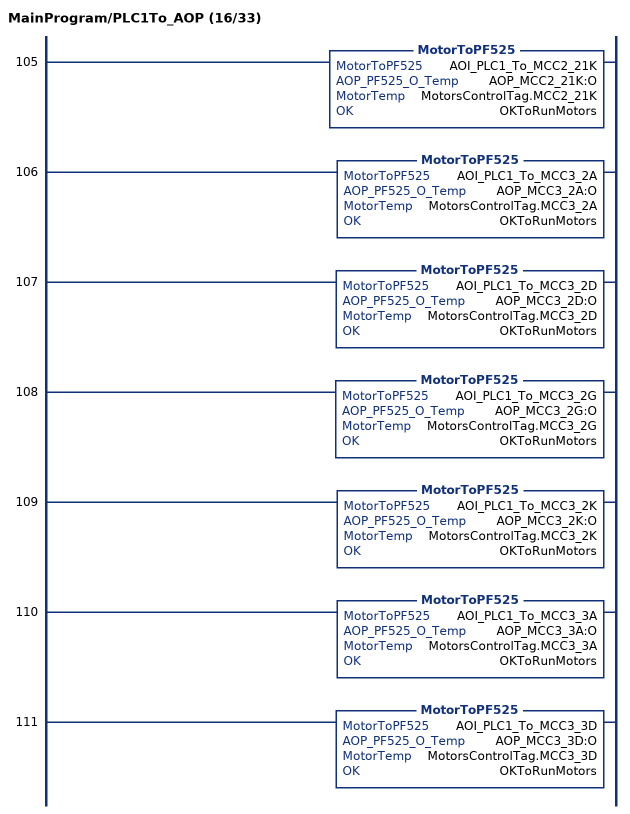
   105: MotorToPF525(AOI_PLC1_To_MCC2_21K,AOP_MCC2_21K:O,MotorsControlTag.MCC2_21K,OKToRunMotors);
   106: MotorToPF525(AOI_PLC1_To_MCC3_2A,AOP_MCC3_2A:O,MotorsControlTag.MCC3_2A,OKToRunMotors);
   107: MotorToPF525(AOI_PLC1_To_MCC3_2D,AOP_MCC3_2D:O,MotorsControlTag.MCC3_2D,OKToRunMotors);
   108: MotorToPF525(AOI_PLC1_To_MCC3_2G,AOP_MCC3_2G:O,MotorsControlTag.MCC3_2G,OKToRunMotors);
   109: MotorToPF525(AOI_PLC1_To_MCC3_2K,AOP_MCC3_2K:O,MotorsControlTag.MCC3_2K,OKToRunMotors);
   110: MotorToPF525(AOI_PLC1_To_MCC3_3A,AOP_MCC3_3A:O,MotorsControlTag.MCC3_3A,OKToRunMotors);
   111: MotorToPF525(AOI_PLC1_To_MCC3_3D,AOP_MCC3_3D:O,MotorsControlTag.MCC3_3D,OKToRunMotors);
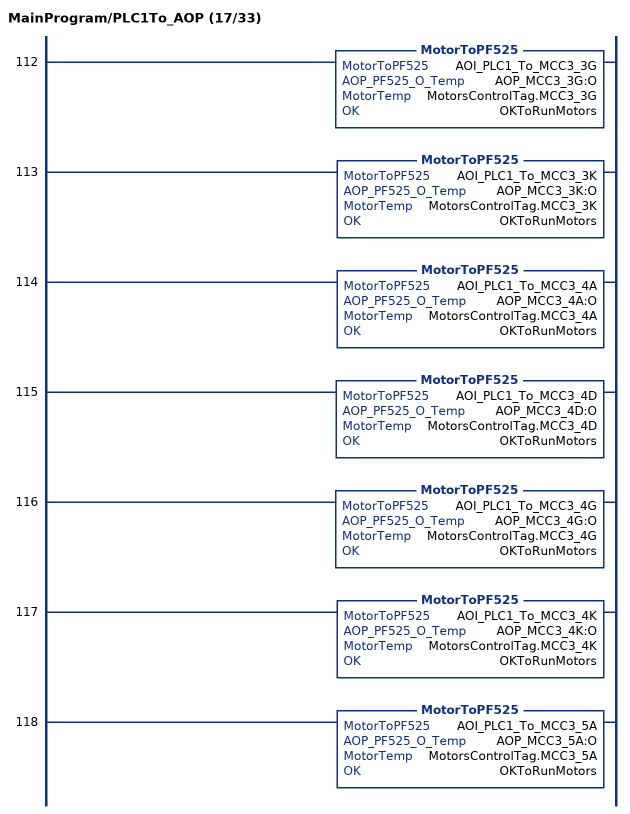
   112: MotorToPF525(AOI_PLC1_To_MCC3_3G,AOP_MCC3_3G:O,MotorsControlTag.MCC3_3G,OKToRunMotors);
   113: MotorToPF525(AOI_PLC1_To_MCC3_3K,AOP_MCC3_3K:O,MotorsControlTag.MCC3_3K,OKToRunMotors);
   114: MotorToPF525(AOI_PLC1_To_MCC3_4A,AOP_MCC3_4A:O,MotorsControlTag.MCC3_4A,OKToRunMotors);
   115: MotorToPF525(AOI_PLC1_To_MCC3_4D,AOP_MCC3_4D:O,MotorsControlTag.MCC3_4D,OKToRunMotors);
   116: MotorToPF525(AOI_PLC1_To_MCC3_4G,AOP_MCC3_4G:O,MotorsControlTag.MCC3_4G,OKToRunMotors);
   117: MotorToPF525(AOI_PLC1_To_MCC3_4K,AOP_MCC3_4K:O,MotorsControlTag.MCC3_4K,OKToRunMotors);
   118: MotorToPF525(AOI_PLC1_To_MCC3_5A,AOP_MCC3_5A:O,MotorsControlTag.MCC3_5A,OKToRunMotors);
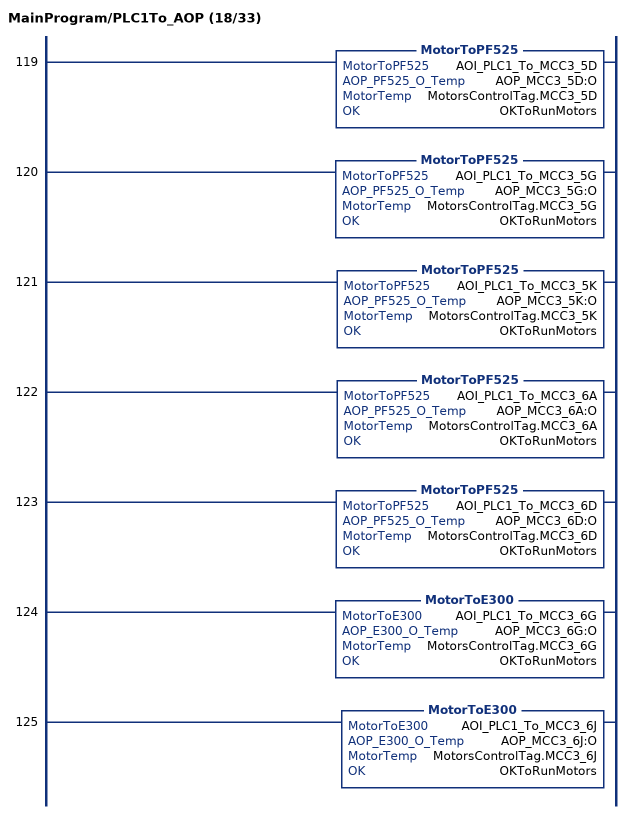
   119: MotorToPF525(AOI_PLC1_To_MCC3_5D,AOP_MCC3_5D:O,MotorsControlTag.MCC3_5D,OKToRunMotors);
   120: MotorToPF525(AOI_PLC1_To_MCC3_5G,AOP_MCC3_5G:O,MotorsControlTag.MCC3_5G,OKToRunMotors);
   121: MotorToPF525(AOI_PLC1_To_MCC3_5K,AOP_MCC3_5K:O,MotorsControlTag.MCC3_5K,OKToRunMotors);
   122: MotorToPF525(AOI_PLC1_To_MCC3_6A,AOP_MCC3_6A:O,MotorsControlTag.MCC3_6A,OKToRunMotors);
   123: MotorToPF525(AOI_PLC1_To_MCC3_6D,AOP_MCC3_6D:O,MotorsControlTag.MCC3_6D,OKToRunMotors);
   124: MotorToE300(AOI_PLC1_To_MCC3_6G,AOP_MCC3_6G:O,MotorsControlTag.MCC3_6G,OKToRunMotors);
   125: MotorToE300(AOI_PLC1_To_MCC3_6J,AOP_MCC3_6J:O,MotorsControlTag.MCC3_6J,OKToRunMotors);
